{attribute 'TcGenerated'}
{attribute 'no-analysis'}
{attribute 'linkalways'}
// This function has been automatically generated from the project information.
VAR_GLOBAL CONSTANT
	{attribute 'const_non_replaced'}
	stLibVersion_TcDeviceBase : ST_LibVersion := (iMajor := 2, iMinor := 0, iBuild := 0, iRevision := 0, nFlags := 0, sVersion := '2.0.0');
END_VAR

(* stored: Version 1.1.0.1, ProductVersion 3.1.4026.13
   GVL Global_Version: Id {91ebc8f1-c017-420b-b63c-f24e63c0f3ee} *)
